FUNCTION_BLOCK FB_SampleListener EXTENDS FB_ListenerBase2
VAR_OUTPUT
		nAlarms	: INT;
END_VAR

METHOD OnAlarmRaised : HRESULT
VAR_INPUT
	fbEvent	: REFERENCE TO FB_TcEvent;
END_VAR
nAlarms := nAlarms+1;
END_METHOD

END_FUNCTION_BLOCK

(* stored: Version 1.1.0.1, ProductVersion 3.1.4024.11
   POU FB_SampleListener: Id {bd686090-6f59-08cd-2ea1-a60d85597367}, SpecialFunc None
   Method OnAlarmRaised: Id {22af7b33-730b-0eb5-3e7e-eb19d892f983} *)
